FUNCTION_BLOCK ButtonNC IMPLEMENTS I_Button
VAR
	bInput	AT%I*	: BOOL;
	rtInput			: R_TRIG;
END_VAR

PROPERTY IsPressed : BOOL
GET
IsPressed := NOT bInput;
END_GET
END_PROPERTY

PROPERTY IsReleased : BOOL
GET
IsReleased := NOT IsPressed;
END_GET
END_PROPERTY

PROPERTY RisingTrigger : BOOL
GET
rtInput(CLK := IsPressed);

RisingTrigger := rtInput.Q;
END_GET
END_PROPERTY

END_FUNCTION_BLOCK

(* stored: Version 1.1.0.1
   POU ButtonNC: Id {da357938-2c55-49d2-ba2f-8a771a077471}, SpecialFunc None
   Property IsPressed: Id {0a66708b-5b01-4a9b-ae62-0f65456f2d04}
   Get Get: Id {18b6dc50-df16-49ca-9718-c45006b8f1b4}
   Property IsReleased: Id {b65fba39-4730-4eab-9747-9da7dcb91829}
   Get Get: Id {53f7de75-988a-4e42-8c0f-a07c837870e3}
   Property RisingTrigger: Id {cbfbe90a-e385-4624-af03-1bb36c4f2056}
   Get Get: Id {866736ee-d9b7-4163-939b-e9443a1f06b9} *)
